{attribute 'GeneratedUsingTerminal: EL3681-0000-0021'}
{attribute addProperty BoxType "EL3681-0000-0021"}
{attribute addProperty Id "SAI_InputsAT %I*SAI_Inputs_84B29FE914SAI_FeedbackAT %I*SAI_Feedback_BDBF6DA92SAI_RangeAT %Q*SAI_Range_2A187FC54WcStateAT %I*WcState_9091E0EB2InfoDataAT %I*InfoData_94A18F5E2"}
{attribute addProperty CRC "2436338260"}
{attribute addProperty Size "24"}
TYPE EL3681_91379254 EXTENDS EtcSlaveTerminalBase_947E5A46 :
STRUCT
	{attribute addProperty Name "SAI_Inputs"}
	SAI_Inputs : SAI_Inputs_84B29FE9;
	{attribute addProperty Name "SAI_Feedback"}
	SAI_Feedback : SAI_Feedback_BDBF6DA9;
	{attribute addProperty Name "SAI_Range"}
	SAI_Range : SAI_Range_2A187FC5;
	{attribute addProperty Name "WcState"}
	WcState : WcState_9091E0EB;
	{attribute addProperty Name "InfoData"}
	InfoData : InfoData_94A18F5E;
END_STRUCT
END_TYPE

(* stored: Version 1.2.0.0, ProductVersion 3.1.4024.9
   DUT EL3681_91379254: Id {b00a4c56-0c5e-44ff-bd8b-e1ed01951e4e} *)
